FUNCTION_BLOCK ULIntComparer EXTENDS Object IMPLEMENTS IComparer
VAR
	_ClassName : STRING := __POUNAME();
END_VAR

{attribute 'monitoring' := 'call'}
PROPERTY ClassName : STRING
GET
ClassName := _ClassName;
END_GET
END_PROPERTY

{attribute "object_name" := "Compare"}
METHOD Compare : COMPARISION_RESULT
VAR_INPUT
	left : __SYSTEM.AnyType;
	right : __SYSTEM.AnyType;
END_VAR
VAR
	leftPointer : POINTER TO ULINT; 
	rightPointer : POINTER TO ULINT; 
END_VAR
IF left.pValue = 0 AND right.pValue = 0 THEN
	Compare := COMPARISION_RESULT.FIRST_EQUAL_TO_SECOND;
	RETURN;
END_IF

IF left.pValue = 0 THEN
	Compare := COMPARISION_RESULT.FIRST_LESS_THAN_SECOND;
	RETURN;	
END_IF

IF right.pValue = 0 THEN
	Compare := COMPARISION_RESULT.FIRST_GREATER_THAN_SECOND;
	RETURN;	
END_IF

leftPointer := left.pValue;
rightPointer := right.pValue;

IF leftPointer^ < rightPointer^ THEN
	Compare := COMPARISION_RESULT.FIRST_LESS_THAN_SECOND;
ELSIF leftPointer^ > rightPointer^ THEN
	Compare := COMPARISION_RESULT.FIRST_GREATER_THAN_SECOND;
ELSE
	Compare := COMPARISION_RESULT.FIRST_EQUAL_TO_SECOND;	
END_IF
END_METHOD

{attribute 'monitoring' := 'call'}
PROPERTY Size : ULINT
GET
Size := XSIZEOF(THIS^);
END_GET
END_PROPERTY

END_FUNCTION_BLOCK

(* stored: Version 1.1.0.1
   POU ULIntComparer: Id {abb0af5d-1df1-4bbf-80af-72605784a464}, SpecialFunc None
   Property ClassName: Id {0d783890-7154-4c86-870a-74c7095fa8fc}
   Get Get: Id {5bc8732b-0287-4375-aecb-23f3fe7a8e64}
   Method Compare: Id {231228dc-138a-495e-91d8-50c0e500507a}
   Property Size: Id {79ff0301-b5cd-4bae-b7cc-6997e735af9d}
   Get Get: Id {1c5f473b-f3dd-44a7-8ce1-6896420c4dad} *)
